// TIA Portal V20 export
TYPE "OPC_SystemStatus"
// stored: Namespace ProductionLine
   STRUCT
      SourceSeq : Int;
   END_STRUCT;
END_TYPE
